// Mitsubishi GX Works2 project: 타이머 예제 1_2   PLC: Q03UDV

PROGRAM MAIN
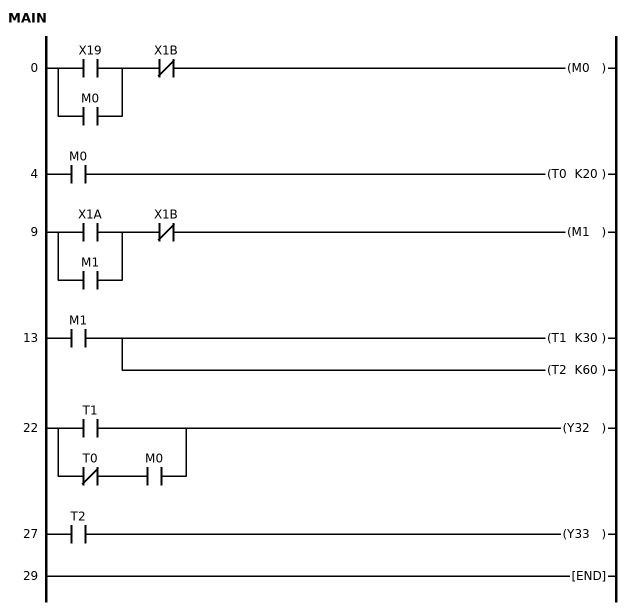
0     LD      X19
      OR      M0
      ANI     X1B
      OUT     M0
4     LD      M0
      OUT     T0 K20
9     LD      X1A
      OR      M1
      ANI     X1B
      OUT     M1
13    LD      M1
      OUT     T1 K30
      OUT     T2 K60
22    LD      T1
      LDI     T0
      AND     M0
      ORB
      OUT     Y32
27    LD      T2
      OUT     Y33
29    END
END_PROGRAM
